% RSLogix 500 project LAB1_BAW.RSS, saved by version 8.40.00.08 %
PROJECT "LAB1_BAW"    % processor: SLC 500, 1747-L541 %

PROGRAM FILES
  LAD 2   8 rungs

DATA FILES
  O0 OUTPUT  68 elements
  I1 INPUT  68 elements
  S2 STATUS  164 elements
  B3 BINARY  1 elements
  T4 TIMER  1 elements
  C5 COUNTER  1 elements
  R6 CONTROL  1 elements
  N7 INTEGER  1 elements
  F8 FLOAT  1 elements

LADDER 2
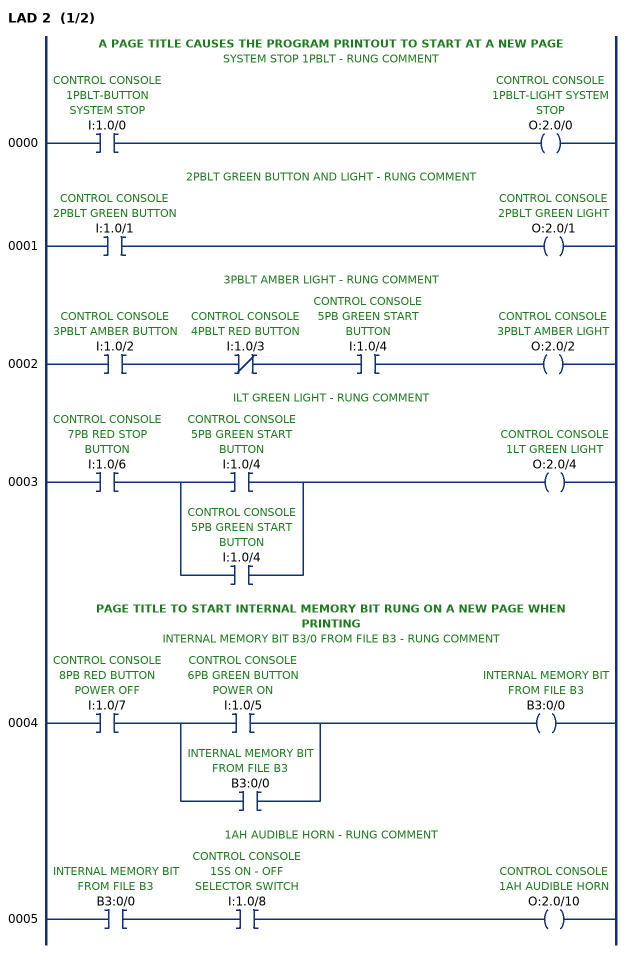
% Rung: 0 %
% TITLE: A PAGE TITLE CAUSES THE PROGRAM PRINTOUT TO START AT A NEW PAGE %
% SYSTEM STOP 1PBLT - RUNG COMMENT %
SOR XIC I:1.0/0 OTE O:2.0/0 EOR
%   I:1.0/0  "CONTROL CONSOLE 1PBLT-BUTTON SYSTEM STOP" %
%   O:2.0/0  "CONTROL CONSOLE 1PBLT-LIGHT SYSTEM STOP" %
% Rung: 1 %
% 2PBLT GREEN BUTTON AND LIGHT - RUNG COMMENT %
SOR XIC I:1.0/1 OTE O:2.0/1 EOR
%   I:1.0/1  "CONTROL CONSOLE 2PBLT GREEN BUTTON" %
%   O:2.0/1  "CONTROL CONSOLE 2PBLT GREEN LIGHT" %
% Rung: 2 %
% 3PBLT AMBER LIGHT - RUNG COMMENT %
SOR XIC I:1.0/2 XIO I:1.0/3 XIC I:1.0/4 OTE O:2.0/2 EOR
%   I:1.0/2  "CONTROL CONSOLE 3PBLT AMBER BUTTON" %
%   I:1.0/3  "CONTROL CONSOLE 4PBLT RED BUTTON" %
%   I:1.0/4  "CONTROL CONSOLE 5PB GREEN START BUTTON" %
%   O:2.0/2  "CONTROL CONSOLE 3PBLT AMBER LIGHT" %
% Rung: 3 %
% ILT GREEN LIGHT - RUNG COMMENT %
SOR XIC I:1.0/6 BST XIC I:1.0/4 NXB XIC I:1.0/4 BND OTE O:2.0/4 EOR
%   I:1.0/6  "CONTROL CONSOLE 7PB RED STOP BUTTON" %
%   I:1.0/4  "CONTROL CONSOLE 5PB GREEN START BUTTON" %
%   O:2.0/4  "CONTROL CONSOLE 1LT GREEN LIGHT" %
% Rung: 4 %
% TITLE: PAGE TITLE TO START INTERNAL MEMORY BIT RUNG ON A NEW PAGE WHEN PRINTING %
% INTERNAL MEMORY BIT B3/0 FROM FILE B3 - RUNG COMMENT %
SOR XIC I:1.0/7 BST XIC I:1.0/5 NXB XIC B3:0/0 BND OTE B3:0/0 EOR
%   I:1.0/7  "CONTROL CONSOLE 8PB RED BUTTON POWER OFF" %
%   I:1.0/5  "CONTROL CONSOLE 6PB GREEN BUTTON POWER ON" %
%   B3:0/0  "INTERNAL MEMORY BIT FROM FILE B3" %
% Rung: 5 %
% 1AH AUDIBLE HORN - RUNG COMMENT %
SOR XIC B3:0/0 XIC I:1.0/8 OTE O:2.0/10 EOR
%   B3:0/0  "INTERNAL MEMORY BIT FROM FILE B3" %
%   I:1.0/8  "CONTROL CONSOLE 1SS ON - OFF SELECTOR SWITCH" %
%   O:2.0/10  "CONTROL CONSOLE 1AH AUDIBLE HORN" %

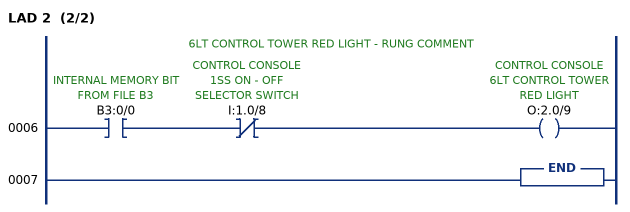
% Rung: 6 %
% 6LT CONTROL TOWER RED LIGHT - RUNG COMMENT %
SOR XIC B3:0/0 XIO I:1.0/8 OTE O:2.0/9 EOR
%   B3:0/0  "INTERNAL MEMORY BIT FROM FILE B3" %
%   I:1.0/8  "CONTROL CONSOLE 1SS ON - OFF SELECTOR SWITCH" %
%   O:2.0/9  "CONTROL CONSOLE 6LT CONTROL TOWER RED LIGHT" %
% Rung: 7 %
SOR END EOR
